// TIA Portal V19 export
VAR_GLOBAL   // PLC tag table "Orchestrator"
END_VAR
